// TwinCAT 3 PLC project PLC1
// ProgramVersion: 3.1.4024.0
// libraries:
//   Tc2_Math, * (Beckhoff Automation GmbH)
//   Tc2_Standard, * (Beckhoff Automation GmbH)
//   Tc2_System, * (Beckhoff Automation GmbH)
//   Tc3_JsonXml, * (Beckhoff Automation GmbH)
//   Tc3_Module, * (Beckhoff Automation GmbH)
// project tree:
//   Common/ AdsLogMessage.TcPOU
//   DynamicArrays/DUTs/ T_DataType.TcDUT
//   DynamicArrays/ DynamicArray.TcCD (not stored), DynamicArrays_Test.TcPOU, FB_DynamicArray.TcPOU, IDynamicArray.TcIO
//   JSON/DomParser/ DomParser.TcCD (not stored), DomParser.TcPOU, FB_DomParserMetaHandler.TcPOU, I_DomParserMetaHandler.TcIO, ST_MetaData.TcDUT
//   OperatorOverloading/CLASS/ FB_Scalar.TcPOU, FB_Vector.TcPOU
//   OperatorOverloading/DUTs/ E_OperatorError.TcDUT
//   OperatorOverloading/ITFs/Core/ I_Object.TcIO, I_Operator.TcIO
//   OperatorOverloading/ITFs/ I_Scalar.TcIO, I_Vector.TcIO
//   OperatorOverloading/ITFs/Operators/ I_Addition.TcIO, I_Division.TcIO, I_Multiplication.TcIO, I_Subtraction.TcIO
//   OperatorOverloading/ OperatorInterafce.TcCD (not stored), OperatorOverloading_Test.TcPOU
//   / PlcTask.TcTTO
//   POUs/ MAIN.TcPOU
// real-time tasks:
//   TASK PlcTask: cycle T#10ms, priority 20, ADS port 350
//   TASK PlcTask1: cycle T#10ms, priority 21, ADS port 351
//   TASK PlcTask2: cycle T#10ms, priority 22, ADS port 352

CONFIGURATION PLC1
    RESOURCE PLC ON TwinCAT3
        TASK PlcTask(INTERVAL := T#10ms, PRIORITY := 20);
        PROGRAM MAIN WITH PlcTask : MAIN;
    END_RESOURCE
END_CONFIGURATION

// ---- DynamicArrays/DUTs/T_DataType.TcDUT
TYPE T_DataType : PVOID; END_TYPE

// ---- JSON/DomParser/ST_MetaData.TcDUT
TYPE ST_MetaData :
STRUCT
  BatteryVoltage : DINT;
  VoltageUnit : STRING;
  ClickType : STRING;
  SensorValue1 : DINT;
END_STRUCT
END_TYPE

// ---- OperatorOverloading/DUTs/E_OperatorError.TcDUT
{attribute 'qualified_only'}
{attribute 'strict'}
{attribute 'to_string'}
TYPE E_OperatorError :
(
	NoError := 0,
	IntegerOverflow := 10,
	NaN,
	PositiveInfinity,
	NegativeInfinity,
	Truncation,
	TypeMismatch := 100
)BYTE;
END_TYPE

// ---- DynamicArrays/IDynamicArray.TcIO
INTERFACE IDynamicArray

METHOD Access : T_DataType
VAR_INPUT
	nPosition : DINT;  // Position of element in dynamic array, 0 indexed.
END_VAR
END_METHOD

METHOD PUBLIC Clear
VAR_INPUT
END_VAR
END_METHOD

METHOD PUBLIC Insert
VAR_INPUT
	Data : T_DataType; // Data to insert in dynamic array.
	nPosition : DINT; // Position to insert data at in the dynamic array, 0 indexed. 
END_VAR
END_METHOD

METHOD PUBLIC IsEmpty : BOOL
VAR_INPUT
END_VAR
END_METHOD

METHOD PUBLIC Resize : BOOL
VAR_INPUT
	nLength 		: DINT; // New length of dynamic array.
END_VAR
END_METHOD

METHOD PUBLIC Show
VAR_IN_OUT
	aList : ARRAY[*] OF T_DataType; // Static array to display data in dynamic array.
END_VAR
END_METHOD

METHOD PUBLIC Size : DINT
VAR_INPUT
END_VAR
END_METHOD

END_INTERFACE

// ---- JSON/DomParser/I_DomParserMetaHandler.TcIO
INTERFACE I_DomParserMetaHandler

PROPERTY BatteryVoltage : DINT
GET
END_GET
END_PROPERTY

METHOD Clear : HRESULT
VAR_INPUT
END_VAR
END_METHOD

PROPERTY ClickType : STRING
GET
END_GET
END_PROPERTY

PROPERTY MetaData : REFERENCE to ST_MetaData
GET
END_GET
END_PROPERTY

PROPERTY SensorValue1 : DINT
GET
END_GET
END_PROPERTY

PROPERTY VoltageUnit : STRING
GET
END_GET
END_PROPERTY

END_INTERFACE

// ---- OperatorOverloading/ITFs/Core/I_Object.TcIO
// Base interface for an object.
INTERFACE I_Object EXTENDS __SYSTEM.IQueryInterface

END_INTERFACE

// ---- OperatorOverloading/ITFs/Core/I_Operator.TcIO
// Base interface for an operator.
INTERFACE I_Operator EXTENDS I_Object

END_INTERFACE

// ---- OperatorOverloading/ITFs/I_Scalar.TcIO
INTERFACE I_Scalar EXTENDS I_Object

METHOD ToF64 : LREAL
VAR_OUTPUT
	e : E_OperatorError;
END_VAR
END_METHOD

METHOD ToI64 : LINT
VAR_OUTPUT
	e : E_OperatorError;
END_VAR
END_METHOD

METHOD ToU8 : BYTE
VAR_OUTPUT
	e : E_OperatorError;
END_VAR
END_METHOD

END_INTERFACE

// ---- OperatorOverloading/ITFs/I_Vector.TcIO
INTERFACE I_Vector EXTENDS I_Object

METHOD ToArray : ARRAY[0..2] OF LREAL
VAR_INPUT
END_VAR
END_METHOD

PROPERTY X : LREAL
GET
END_GET
SET
END_SET
END_PROPERTY

PROPERTY Y : LREAL
GET
END_GET
SET
END_SET
END_PROPERTY

PROPERTY Z : LREAL
GET
END_GET
SET
END_SET
END_PROPERTY

END_INTERFACE

// ---- OperatorOverloading/ITFs/Operators/I_Addition.TcIO
INTERFACE I_Addition EXTENDS I_Operator

METHOD Plus : I_Addition
VAR_INPUT
	ipObject : I_Object;
END_VAR
VAR_OUTPUT
	e : E_OperatorError;
END_VAR
END_METHOD

END_INTERFACE

// ---- OperatorOverloading/ITFs/Operators/I_Division.TcIO
INTERFACE I_Division EXTENDS I_Operator

METHOD DivideBy : I_Division
VAR_INPUT
	ipObject : I_Object;
END_VAR
VAR_OUTPUT
	e : E_OperatorError;
END_VAR
END_METHOD

END_INTERFACE

// ---- OperatorOverloading/ITFs/Operators/I_Multiplication.TcIO
INTERFACE I_Multiplication EXTENDS I_Operator

METHOD Times : I_Multiplication
VAR_INPUT
	ipObject : I_Object;
END_VAR
VAR_OUTPUT
	e : E_OperatorError;
END_VAR
END_METHOD

END_INTERFACE

// ---- OperatorOverloading/ITFs/Operators/I_Subtraction.TcIO
INTERFACE I_Subtraction EXTENDS I_Operator

METHOD Minus : I_Subtraction
VAR_INPUT
	ipObject : I_Object;
END_VAR
VAR_OUTPUT
	e : E_OperatorError;
END_VAR
END_METHOD

END_INTERFACE

// ---- POUs/MAIN.TcPOU
PROGRAM MAIN
VAR
END_VAR


DomParser();
OperatorOverloading_Test();
DynamicArrays_Test();

END_PROGRAM

// ---- JSON/DomParser/DomParser.TcPOU
PROGRAM DomParser
VAR
  
  sMessage : T_MAXSTRING := '{"serialNumber":"123","meta":{"batteryVoltage":"1547", "voltageUnit" : "mV", "clickType":"SINGLE", "sensorValue1" : 3462}}';
  fbJson : Tc3_JsonXml.FB_JsonDomParser;
  jsonIterator : SJsonIterator;
  jsonIteratorEnd : SJsonIterator;
  
  jsonDoc : SJsonValue;
  sName : T_MAXSTRING;
  jsonValue : SJsonValue;
  sMetaData : T_MAXSTRING; //{"batteryVoltage":"1547", "voltageUnit" : "mV", "clickType":"SINGLE", "sensorValue1" : 3462} 
  bGetMetaData : BOOL;
  
END_VAR
VAR
  // parsen
 	fbJsonParser : FB_JsonSaxReader;
  pDomParserMetaHandler : FB_DomParserMetaHandler;
  iMetaData : I_DomParserMetaHandler := pDomParserMetaHandler;
  stMetaData : ST_MetaData;

END_VAR


// CopyJson()

jsonDoc         := fbJson.ParseDocument(sMessage);
jsonIterator    := fbJson.MemberBegin(jsonDoc);
jsonIteratorEnd := fbJson.MemberEnd(jsonDoc);

IF bGetMetaData THEN
  WHILE jsonIterator <> jsonIteratorEnd DO
    sName         := fbJson.GetMemberName(jsonIterator);
    jsonValue     := fbJson.GetMemberValue(jsonIterator);
    IF sName = 'meta' THEN
      fbJson.CopyJson(jsonValue, sMetaData, SIZEOF(sMetaData));
      fbJsonParser.ParseValues(sMetaData, pDomParserMetaHandler);
      bGetMetaData := FALSE;
      EXIT;
      END_IF
    jsonIterator  := fbJson.NextMember(jsonIterator);
    END_WHILE
  END_IF

  stMetaData.BatteryVoltage := iMetaData.MetaData.BatteryVoltage;

END_PROGRAM

// ---- JSON/DomParser/FB_DomParserMetaHandler.TcPOU
//{attribute 'hide_all_locals'}
{attribute 'c++_compatible'}
FUNCTION_BLOCK PUBLIC FB_DomParserMetaHandler IMPLEMENTS ITcJsonSaxValues, I_DomParserMetaHandler
VAR_INPUT
END_VAR
VAR_OUTPUT
END_VAR
VAR
  // Properties
  _batteryVoltage : DINT;
  _voltageUnit : STRING;
  _clickType : STRING;
  _sensorValue1 : DINT;
  _metaData : ST_MetaData;

END_VAR

{warning 'Eigenschaftenimplementierung hinzufügen'}
PROPERTY BatteryVoltage : DINT
GET

BatteryVoltage := THIS^._batteryVoltage;
END_GET
END_PROPERTY


METHOD Clear : HRESULT

THIS^._batteryVoltage := 0;
THIS^._sensorValue1 := 0;
THIS^._clickType := '';
THIS^._voltageUnit := '';

Clear := Tc3_Module.S_OK;
END_METHOD


PROPERTY ClickType : STRING
GET

ClickType := THIS^._clickType;
END_GET
END_PROPERTY


PROPERTY MetaData : REFERENCE TO ST_MetaData
GET

MetaData REF= _metaData;
END_GET
END_PROPERTY

{attribute 'TcTypeSystem'}
{attribute 'no-analysis'}
{attribute 'c++_compatible'}
{attribute 'minimal_input_size' := '4'}
{attribute 'pack_mode' := '4'}
METHOD OnBoolValue : HRESULT
VAR_INPUT
	level	: UDINT;
	infos	: POINTER TO TcJsonLevelInfo;
	value	: BOOL;
END_VAR

AdsLogMessage('OnBoolValue');

OnBoolValue := Tc3_Module.S_OK;
END_METHOD

{attribute 'TcTypeSystem'}
{attribute 'no-analysis'}
{attribute 'c++_compatible'}
{attribute 'minimal_input_size' := '4'}
{attribute 'pack_mode' := '4'}
METHOD OnDintValue : HRESULT
VAR_INPUT
	level	: UDINT;
	infos	: POINTER TO TcJsonLevelInfo;
	value	: DINT;
END_VAR

AdsLogMessage('OnDintValue');

OnDintValue := Tc3_Module.S_OK;
END_METHOD

{attribute 'TcTypeSystem'}
{attribute 'no-analysis'}
{attribute 'c++_compatible'}
{attribute 'minimal_input_size' := '4'}
{attribute 'pack_mode' := '4'}
METHOD OnLintValue : HRESULT
VAR_INPUT
	level	: UDINT;
	infos	: POINTER TO TcJsonLevelInfo;
	value	: LINT;
END_VAR

AdsLogMessage('OnLintValue');

OnLintValue := Tc3_Module.S_OK;
END_METHOD

{attribute 'TcTypeSystem'}
{attribute 'no-analysis'}
{attribute 'c++_compatible'}
{attribute 'minimal_input_size' := '4'}
{attribute 'pack_mode' := '4'}
METHOD OnLrealValue : HRESULT
VAR_INPUT
	level	: UDINT;
	infos	: POINTER TO TcJsonLevelInfo;
	value	: LREAL;
END_VAR

AdsLogMessage('OnLrealValue');

OnLrealValue := Tc3_Module.S_OK;
END_METHOD

{attribute 'TcTypeSystem'}
{attribute 'no-analysis'}
{attribute 'c++_compatible'}
{attribute 'minimal_input_size' := '4'}
{attribute 'pack_mode' := '4'}
METHOD OnNullValue : HRESULT
VAR_INPUT
	level	: UDINT;
	infos	: POINTER TO TcJsonLevelInfo;
END_VAR

AdsLogMessage('OnNullValue');

OnNullValue := Tc3_Module.S_OK;
END_METHOD

{attribute 'TcTypeSystem'}
{attribute 'no-analysis'}
{attribute 'c++_compatible'}
{attribute 'minimal_input_size' := '4'}
{attribute 'pack_mode' := '4'}
METHOD OnRawNumberValue : HRESULT
VAR_INPUT
	level	: UDINT;
	infos	: POINTER TO TcJsonLevelInfo;
END_VAR
VAR_IN_OUT CONSTANT
	value	: STRING;
END_VAR
VAR_INPUT
	len	: UDINT;
END_VAR

AdsLogMessage('OnRawNumberValue');

OnRawNumberValue := Tc3_Module.S_OK;
END_METHOD

{attribute 'TcTypeSystem'}
{attribute 'no-analysis'}
{attribute 'c++_compatible'}
{attribute 'minimal_input_size' := '4'}
{attribute 'pack_mode' := '4'}
METHOD OnStringValue : HRESULT
VAR_INPUT
	level	: UDINT;
	infos	: POINTER TO TcJsonLevelInfo;
END_VAR
VAR_IN_OUT CONSTANT
	value	: STRING;
END_VAR
VAR_INPUT
	len	: UDINT;
END_VAR

AdsLogMessage('OnStringValue');

SetData(level, infos^, value);

OnStringValue := Tc3_Module.S_OK;
END_METHOD

{attribute 'TcTypeSystem'}
{attribute 'no-analysis'}
{attribute 'c++_compatible'}
{attribute 'minimal_input_size' := '4'}
{attribute 'pack_mode' := '4'}
METHOD OnUdintValue : HRESULT
VAR_INPUT
	level	: UDINT;
	infos	: POINTER TO TcJsonLevelInfo;
	value	: UDINT;
END_VAR

AdsLogMessage('OnUdintValue');

OnUdintValue := Tc3_Module.S_OK;
END_METHOD

{attribute 'TcTypeSystem'}
{attribute 'no-analysis'}
{attribute 'c++_compatible'}
{attribute 'minimal_input_size' := '4'}
{attribute 'pack_mode' := '4'}
METHOD OnUlintValue : HRESULT
VAR_INPUT
	level	: UDINT;
	infos	: POINTER TO TcJsonLevelInfo;
	value	: ULINT;
END_VAR

AdsLogMessage('OnUlintValue');

OnUlintValue := Tc3_Module.S_OK;
END_METHOD


PROPERTY SensorValue1 : DINT
GET

SensorValue1 := THIS^._sensorValue1;
END_GET
END_PROPERTY

METHOD PRIVATE SetData : HRESULT
VAR_INPUT
	level	: UDINT;
	infos	: TcJsonLevelInfo;
	value	: STRING;
END_VAR
VAR
  hr : HRESULT;
END_VAR

IF infos.key^ = 'batteryVoltage' THEN
  THIS^._batteryVoltage := TO_DINT(value);
  THIS^._metaData.BatteryVoltage := THIS^._batteryVoltage;

ELSIF infos.key^ = 'voltageUnit' THEN
  THIS^._voltageUnit := value; 
  THIS^._metaData.VoltageUnit := THIS^._voltageUnit;

ELSIF infos.key^ = 'clickType' THEN
  THIS^._clickType := value; 
  THIS^._metaData.ClickType := THIS^._clickType;


ELSIF infos.key^ = 'sensorValue1' THEN
  THIS^._sensorValue1 := TO_DINT(value);
  THIS^._metaData.SensorValue1 := THIS^._sensorValue1;

ELSE
    hr := Tc3_Module.E_FAIL;
  END_IF

SetData := hr;
END_METHOD

{attribute 'TcTypeSystem'}
{attribute 'no-analysis'}
{attribute 'c++_compatible'}
{attribute 'minimal_input_size' := '4'}
{attribute 'pack_mode' := '4'}
{warning 'Methodenimplementierung hinzufügen'}
METHOD TcAddRef : UDINT
END_METHOD

{attribute 'TcTypeSystem'}
{attribute 'no-analysis'}
{attribute 'c++_compatible'}
{attribute 'minimal_input_size' := '4'}
{attribute 'pack_mode' := '4'}
{warning 'Methodenimplementierung hinzufügen'}
METHOD TcQueryInterface : HRESULT
VAR_INPUT
	iid	: REFERENCE TO IID;
	pipItf	: POINTER TO PVOID;
END_VAR
END_METHOD

{attribute 'TcTypeSystem'}
{attribute 'no-analysis'}
{attribute 'c++_compatible'}
{attribute 'minimal_input_size' := '4'}
{attribute 'pack_mode' := '4'}
{warning 'Methodenimplementierung hinzufügen'}
METHOD TcRelease : UDINT
END_METHOD


PROPERTY VoltageUnit : STRING
GET

VoltageUnit := THIS^._voltageUnit;
END_GET
END_PROPERTY

END_FUNCTION_BLOCK

// ---- Common/AdsLogMessage.TcPOU
FUNCTION AdsLogMessage : BOOL
VAR_INPUT
  sMessage : STRING;
END_VAR
VAR
  sMsgFormat : STRING := 'PLC Msg: %s';
  msgCtrlMask : DWORD := ADSLOG_MSGTYPE_HINT OR ADSLOG_MSGTYPE_LOG;
END_VAR


ADSLOGSTR(msgCtrlMask:= msgCtrlMask, msgFmtStr:= sMsgFormat, strArg:= sMessage);

END_FUNCTION

// ---- OperatorOverloading/OperatorOverloading_Test.TcPOU

// Lib: Tc2_Math

PROGRAM OperatorOverloading_Test
VAR
	bDoubleSquareScal, bAddVec, bCrossProd, bScaleVec : BOOL;
	eError : E_OperatorError;
	fbScalar : FB_Scalar(2.2);
	fbVector1 : FB_Vector(1,2,3);
	fbVector2 : FB_Vector(3,2,1);
END_VAR


// Direkt
IF bDoubleSquareScal THEN 
	bDoubleSquareScal := FALSE;
	fbScalar.Times(fbScalar.Plus(fbScalar));
	END_IF

IF bAddVec THEN
	bAddVec := FALSE;
	fbVector1.Plus(fbVector2);
	END_IF
	
IF bCrossProd THEN
	bCrossProd := FALSE;
	fbVector1.Times(fbVector2);
	END_IF
	
IF bScaleVec THEN
	bScaleVec := FALSE;
	fbVector1.Times(fbScalar);
	END_IF

END_PROGRAM

// ---- OperatorOverloading/CLASS/FB_Scalar.TcPOU
{attribute 'no_explicit_call' := 'do not call this function block directly'}
FUNCTION_BLOCK FB_Scalar IMPLEMENTS I_Scalar, I_Addition, I_Subtraction, I_Multiplication, I_Division
VAR
	_fValue : LREAL; 
END_VAR

METHOD DivideBy : I_Division
VAR_INPUT
	ipObject : I_Object;
END_VAR
VAR_OUTPUT
	e : E_OperatorError;
END_VAR
VAR
	Tmp : LREAL;
	ipNumber : I_Scalar;
END_VAR
DivideBy := THIS^;

IF NOT __QUERYINTERFACE(ipObject, ipNumber) THEN e := E_OperatorError.TypeMismatch; RETURN; END_IF

Tmp := ipNumber.ToF64(e => e);
IF Tmp = 0 THEN 
	THIS^._fValue := SEL(Tmp > 0, -1*TO_LREAL('#Inf'), TO_LREAL('#Inf'));
	RETURN;
	END_IF

IF e <> E_OperatorError.NoError THEN 
	THIS^._fValue := ipNumber.ToF64();
	END_IF

THIS^._fValue := THIS^.ToF64() / ipNumber.ToF64();
END_METHOD

{attribute 'hide'}
METHOD FB_init : BOOL
VAR_INPUT
	bInitRetains : BOOL; // if TRUE, the retain variables are initialized (warm start / cold start)
	bInCopyCode : BOOL;  // if TRUE, the instance afterwards gets moved into the copy code (online change)
	fInitValue : LREAL;
END_VAR
THIS^._fValue := fInitValue;
END_METHOD

METHOD Minus : I_Subtraction
VAR_INPUT
	ipObject : I_Object;
END_VAR
VAR_OUTPUT
	e : E_OperatorError;
END_VAR
VAR
	e1, e2 : E_OperatorError;
	ipNumber : I_Scalar;
END_VAR
Minus := THIS^;

IF NOT __QUERYINTERFACE(ipObject, ipNumber) THEN
  e := E_OperatorError.TypeMismatch; 
  RETURN;
  END_IF

THIS^._fValue := THIS^.ToF64(e => e1) - ipNumber.ToF64(e => e2);

e := MAX(e1, e2);
END_METHOD

METHOD Plus : I_Addition
VAR_INPUT
	ipObject : I_Object;
END_VAR
VAR_OUTPUT
	e : E_OperatorError;
END_VAR
VAR
	e1, e2 : E_OperatorError;
	ipNumber : I_Scalar;
END_VAR
Plus := THIS^;

IF NOT __QUERYINTERFACE(ipObject, ipNumber) THEN e := E_OperatorError.TypeMismatch; RETURN; END_IF

THIS^._fValue := THIS^.ToF64(e => e1) + ipNumber.ToF64(e => e2);

e := MAX(e1, e2);
END_METHOD

METHOD SetValue : REFERENCE TO FB_Scalar
VAR_INPUT
	fValue : LREAL;
END_VAR
SetValue REF= THIS^;

THIS^._fValue := fValue;
END_METHOD

METHOD Times : I_Multiplication
VAR_INPUT
	ipObject : I_Object;
END_VAR
VAR_OUTPUT
	e : E_OperatorError;
END_VAR
VAR
	e1, e2 : E_OperatorError;
	ipNumber : I_Scalar;
END_VAR
Times := THIS^;

IF NOT __QUERYINTERFACE(ipObject, ipNumber) THEN e := E_OperatorError.TypeMismatch; RETURN; END_IF

THIS^._fValue := THIS^.ToF64(e => e1) * ipNumber.ToF64( e => e2);

e := MAX(e1, e2);
END_METHOD

METHOD ToF64 : LREAL
VAR_OUTPUT
	e	: E_OperatorError;
END_VAR
ToF64 := THIS^._fValue;

IF TO_STRING(THIS^._fValue) = '#NaN' THEN 
	e := E_OperatorError.NaN;
ELSIF TO_STRING(THIS^._fValue) = '#Inf' THEN
	e := E_OperatorError.PositiveInfinity;
ELSIF TO_STRING(THIS^._fValue) = '-#Inf' THEN
	e := E_OperatorError.NegativeInfinity;
	END_IF
END_METHOD

METHOD ToI64 : LINT
VAR_OUTPUT
	e	: E_OperatorError;
END_VAR
ToI64 := TO_LINT(THIS^._fValue);

// Check for truncation.
IF Tc2_Math.FRAC(THIS^._fValue) <> 0  THEN 
	e := E_OperatorError.Truncation;
	END_IF
END_METHOD

METHOD ToU8 : BYTE
VAR_OUTPUT
	e	: E_OperatorError;
END_VAR
ToU8 := TO_BYTE(THIS^._fValue);

// Check for truncation.
IF Tc2_Math.FRAC(THIS^._fValue) <> 0  THEN 
	e := E_OperatorError.Truncation;
	END_IF

// Bounds check.
IF THIS^._fValue < 0 OR THIS^._fValue > 255 THEN 
	e := E_OperatorError.IntegerOverflow;
	END_IF
END_METHOD

END_FUNCTION_BLOCK

// ---- OperatorOverloading/CLASS/FB_Vector.TcPOU
{attribute 'no_explicit_call' := 'do not call this function block directly'}
FUNCTION_BLOCK FB_Vector IMPLEMENTS I_Vector, I_Addition, I_Subtraction, I_Multiplication
VAR
	_fX, _fY, _fZ : LREAL;
END_VAR

{attribute 'hide'}
METHOD FB_init : BOOL
VAR_INPUT
	bInitRetains : BOOL; // if TRUE, the retain variables are initialized (warm start / cold start)
	bInCopyCode : BOOL;  // if TRUE, the instance afterwards gets moved into the copy code (online change)
	fX, fY, fZ : LREAL;
END_VAR
THIS^.SetValue(fX, fY, fZ);
END_METHOD

METHOD Minus : I_Subtraction
VAR_INPUT
	ipObject : I_Object;
END_VAR
VAR_OUTPUT
	e : E_OperatorError;
END_VAR
VAR
	ipVector : I_Vector;
END_VAR
Minus := THIS^;

IF NOT __QUERYINTERFACE(ipObject, ipVector) THEN
  e := E_OperatorError.TypeMismatch;
  RETURN;
  END_IF

THIS^._fX := THIS^._fX - ipVector.X;
THIS^._fY := THIS^._fY - ipVector.Y;
THIS^._fZ := THIS^._fZ - ipVector.Z;
END_METHOD

METHOD Plus : I_Addition
VAR_INPUT
	ipObject : I_Object;
END_VAR
VAR_OUTPUT
	e : E_OperatorError;
END_VAR
VAR
	ipVector : I_Vector;
END_VAR
Plus := THIS^;

IF NOT __QUERYINTERFACE(ipObject, ipVector) THEN
  e := E_OperatorError.TypeMismatch; 
  RETURN;
  END_IF

THIS^._fX := THIS^._fX + ipVector.X;
THIS^._fY := THIS^._fY + ipVector.Y;
THIS^._fZ := THIS^._fZ + ipVector.Z;
END_METHOD

METHOD SetValue : REFERENCE TO FB_Vector
VAR_INPUT
	fX, fY, fZ : LREAL;
END_VAR
SetValue REF= THIS^;

THIS^._fX := fX;
THIS^._fY := fY;
THIS^._fZ := fZ;
END_METHOD

METHOD Times : I_Multiplication
VAR_INPUT
	ipObject : I_Object;
END_VAR
VAR_OUTPUT
	e : E_OperatorError;
END_VAR
VAR
	ipNumber : I_Scalar;
	ipVector : I_Vector;
	TmpX, TmpY, TmpZ : LREAL;
END_VAR
Times := THIS^;

// Scale vector.
IF __QUERYINTERFACE(ipObject, ipNumber) THEN 
	THIS^.SetValue( THIS^._fX * ipNumber.ToF64(),
					THIS^._fY * ipNumber.ToF64(),
					THIS^._fZ * ipNumber.ToF64());
	RETURN;
	END_IF

// Do the cross-product.
IF __QUERYINTERFACE(ipObject, ipVector) THEN 
	TmpX := THIS^._fX;
  TmpY := THIS^._fY;
  TmpZ := THIS^._fZ;
  
	THIS^.SetValue(	(TmpY*ipVector.Z) - (TmpZ*ipVector.Y),
					        (TmpZ*ipVector.X) - (TmpX*ipVector.Y),
					        (TmpX*ipVector.Y) - (TmpY*ipVector.X));
	
	RETURN; 
	END_IF

e := E_OperatorError.TypeMismatch;
END_METHOD

METHOD ToArray : ARRAY[0..2] OF LREAL
VAR_INPUT
END_VAR

ToArray[0]:= THIS^._fX;
ToArray[1]:= THIS^._fY;
ToArray[2]:= THIS^._fZ;
END_METHOD

PROPERTY X : LREAL
GET
X := THIS^._fX;
END_GET
SET
THIS^._fX := X;
END_SET
END_PROPERTY

PROPERTY Y : LREAL
GET
Y := THIS^._fY;
END_GET
SET
THIS^._fY:= Y;
END_SET
END_PROPERTY

PROPERTY Z : LREAL
GET
Z := THIS^._fZ;
END_GET
SET
THIS^._fZ := Z;
END_SET
END_PROPERTY

END_FUNCTION_BLOCK

// ---- DynamicArrays/DynamicArrays_Test.TcPOU
PROGRAM DynamicArrays_Test
VAR
	bIsEmpty : BOOL;
  bInsert, bAdd, bAccess, bResize, bClear : BOOL;
	nDynamicSize : DINT;
	aArray : ARRAY[0..30] OF T_DataType;
	tAccess : T_DataType;
  
	fbDynamicArray : FB_DynamicArray(10);
  iDynamicArray : IDynamicArray := fbDynamicArray;
  
	nIdx : DINT;
  
END_VAR



// direct Access

//bIsEmpty := fbDynamicArray.IsEmpty();
//nDynamicSize := fbDynamicArray.Size();
//fbDynamicArray.Show(aArray);

//IF bInsert THEN
//	fbDynamicArray.Insert(53476,0); 
//	FOR nIdx := 1 TO 9 DO 
//    fbDynamicArray.Insert(TO_ULINT(nIdx * 11), nIdx);
//    END_FOR
//	bInsert := FALSE;
//	END_IF

//IF bAdd THEN
//  fbDynamicArray.Insert(33,10);
//  bAdd := FALSE;
//  END_IF

//IF bAccess THEN
//  tAccess := fbDynamicArray.Access(2);
//  bAccess := FALSE;
//  END_IF

//IF bResize THEN
//  fbDynamicArray.Resize(5); 
//  bResize := FALSE;
//  END_IF

//IF bClear THEN
//  fbDynamicArray.Clear(); 
//  bClear := FALSE;
//  END_IF

  
  
  
// Interface Access

bIsEmpty := iDynamicArray.IsEmpty();
nDynamicSize := iDynamicArray.Size();
iDynamicArray.Show(aArray);

IF bInsert THEN
	iDynamicArray.Insert(53476,0); 
	FOR nIdx := 1 TO 9 DO 
    iDynamicArray.Insert(TO_ULINT(nIdx * 11), nIdx);
    END_FOR
	bInsert := FALSE;
	END_IF

IF bAdd THEN
  iDynamicArray.Insert(33,10);
  bAdd := FALSE;
  END_IF

IF bAccess THEN
  tAccess := iDynamicArray.Access(2);
  bAccess := FALSE;
  END_IF

IF bResize THEN
  iDynamicArray.Resize(5); 
  bResize := FALSE;
  END_IF

IF bClear THEN
  iDynamicArray.Clear(); 
  bClear := FALSE;
  END_IF

END_PROGRAM

// ---- DynamicArrays/FB_DynamicArray.TcPOU
FUNCTION_BLOCK PUBLIC FB_DynamicArray IMPLEMENTS IDynamicArray
VAR_INPUT
END_VAR
VAR_OUTPUT
END_VAR
VAR
	pData 	: POINTER TO T_DataType;
	nLength : DINT;
	tNull	: T_DataType;
  
END_VAR

METHOD PUBLIC Access : T_DataType
VAR_INPUT
	nPosition : DINT;  // Position of element in dynamic array, 0 indexed.
END_VAR

IF nPosition < 0 THEN
  Access := tNull;
  RETURN;
  END_IF
  
IF THIS^.IsEmpty() THEN
  FB_Init(FALSE,FALSE,(nPosition + 1) * 2);
  END_IF
  
IF nPosition >= THIS^.Size() THEN
  THIS^.Insert(tNull, nPosition);
  END_IF

Access := THIS^.pData[nPosition];
END_METHOD

METHOD PUBLIC Clear
VAR_INPUT
END_VAR

IF NOT(THIS^.IsEmpty()) THEN 
  __DELETE(THIS^.pData); 
  THIS^.IsEmpty();
  END_IF
END_METHOD

METHOD FB_exit : BOOL
VAR_INPUT
	bInCopyCode : BOOL; // if TRUE, the exit method is called for exiting an instance that is copied afterwards (online change).
END_VAR

THIS^.Clear();
END_METHOD

METHOD FB_init : BOOL
VAR_INPUT
	bInitRetains : BOOL; // if TRUE, the retain variables are initialized (warm start / cold start)
	bInCopyCode : BOOL;  // if TRUE, the instance afterwards gets moved into the copy code (online change)
	nLength : DINT; 	// Length to initialize array with, default is 10;
END_VAR

THIS^.Clear();
IF nLength > 0 THEN
  THIS^.pData := __NEW(T_DataType, TO_UDINT(nLength));
  END_IF

THIS^.nLength := nLength;
END_METHOD

METHOD PUBLIC Insert
VAR_INPUT
	Data : T_DataType; // Data to insert in dynamic array.
	nPosition : DINT; // Position to insert data at in the dynamic array, 0 indexed. 
END_VAR
VAR
	pTemp_Data : POINTER TO T_DataType;
	nTemp_Length : DINT;
	i : DINT;
END_VAR

IF nPosition < 0 THEN RETURN; END_IF

IF THIS^.IsEmpty() THEN
  FB_Init(FALSE,FALSE,(nPosition+1)*2);
  END_IF

IF nPosition < THIS^.Size() THEN 
	THIS^.pData[nPosition] := Data;
ELSE 
	THIS^.Resize((nPosition+1)*2);
	THIS^.pData[nPosition] := Data;
	END_IF
END_METHOD

METHOD PUBLIC IsEmpty : BOOL
VAR_INPUT
END_VAR

IsEmpty := THIS^.pData = 0;
IF IsEmpty THEN
  THIS^.nLength := 0; 
  END_IF
END_METHOD

METHOD PUBLIC Resize : BOOL
VAR_INPUT
	nLength 		: DINT; // New length of dynamic array.
END_VAR
VAR_INST
	pOldData : POINTER TO T_DataType;
	nOldLength : DINT;
	nIdx : DINT;
END_VAR


IF nLength <= 0 THEN 
  THIS^.Clear(); 
  RETURN; 
  END_IF

IF THIS^.IsEmpty() THEN
  FB_init(FALSE,FALSE,nLength); 
  RETURN;
  END_IF
  
IF THIS^.nLength = nLength THEN RETURN; END_IF

// save old Data
pOldData 		:= THIS^.pData; 

nOldLength 	:= THIS^.nLength;
THIS^.nLength 	:= nLength;

// allocate new Data
THIS^.pData := __NEW(T_DataType, TO_UDINT(THIS^.nLength));

// copy old Data
FOR nIdx := 0 TO TO_DINT(nOldLength-1) DO 
	IF nIdx > TO_DINT(THIS^.nLength-1) THEN EXIT; END_IF
 
	THIS^.pData[nIdx] := pOldData[nIdx]; 
	END_FOR

// delete old Data
__DELETE(pOldData);
END_METHOD

METHOD PUBLIC Show
VAR_IN_OUT
	aList : ARRAY[*] OF T_DataType; // Static array to display data in dynamic array.
END_VAR
VAR
	nIdx,nIdxData : DINT;
END_VAR

FOR nIdx := LOWER_BOUND(aList, 1) TO UPPER_BOUND(aList, 1) DO
	IF (nIdxData < TO_DINT(THIS^.Size())) AND NOT(THIS^.IsEmpty()) THEN
		aList[nIdx] := THIS^.pData[nIdxData];
		nIdxData := nIdxData + 1; 
	ELSE 
		aList[nIdx] := tNull;
	 	END_IF
	END_FOR
END_METHOD

METHOD PUBLIC Size : DINT
VAR_INPUT
END_VAR

//IsEmpty(); 
Size := THIS^.nLength;
END_METHOD

END_FUNCTION_BLOCK
